{attribute 'GeneratedUsingTerminal: EJ7411-0000-0018'}
{attribute addProperty BoxType "EJ7411-0000-0018"}
{attribute addProperty Id "FB_PositionAT %I*FB_Position_3FA094ED4DRV_StatuswordAT %I*DRV_Statusword_9B36FDFC2DRV_Following_error_actual_valueAT %I*DRV_Following_error_actual_value_5AA320BF4DRV_ControlwordAT %Q*DRV_Controlword_F3F147212DRV_Target_positionAT %Q*DRV_Target_position_05240F144WcStateAT %I*WcState_9091E0EB2InfoDataAT %I*InfoData_0F6C743412"}
{attribute addProperty CRC "3601388696"}
{attribute addProperty Size "30"}
TYPE EJ7411_D6A8D498 EXTENDS EtcSlaveTerminalBase_947E5A46 :
STRUCT
	{attribute addProperty Name "FB_Position"}
	FB_Position : FB_Position_3FA094ED;
	{attribute addProperty Name "DRV_Statusword"}
	DRV_Statusword : DRV_Statusword_9B36FDFC;
	{attribute addProperty Name "DRV_Following_error_actual_value"}
	DRV_Following_error_actual_value : DRV_Following_error_actual_value_5AA320BF;
	{attribute addProperty Name "DRV_Controlword"}
	DRV_Controlword : DRV_Controlword_F3F14721;
	{attribute addProperty Name "DRV_Target_position"}
	DRV_Target_position : DRV_Target_position_05240F14;
	{attribute addProperty Name "WcState"}
	WcState : WcState_9091E0EB;
	{attribute addProperty Name "InfoData"}
	InfoData : InfoData_0F6C7434;
END_STRUCT
END_TYPE

(* stored: Version 1.2.0.0, ProductVersion 3.1.4024.9
   DUT EJ7411_D6A8D498: Id {c20b5aee-d245-4cbe-8ae7-7e4745724e33} *)
